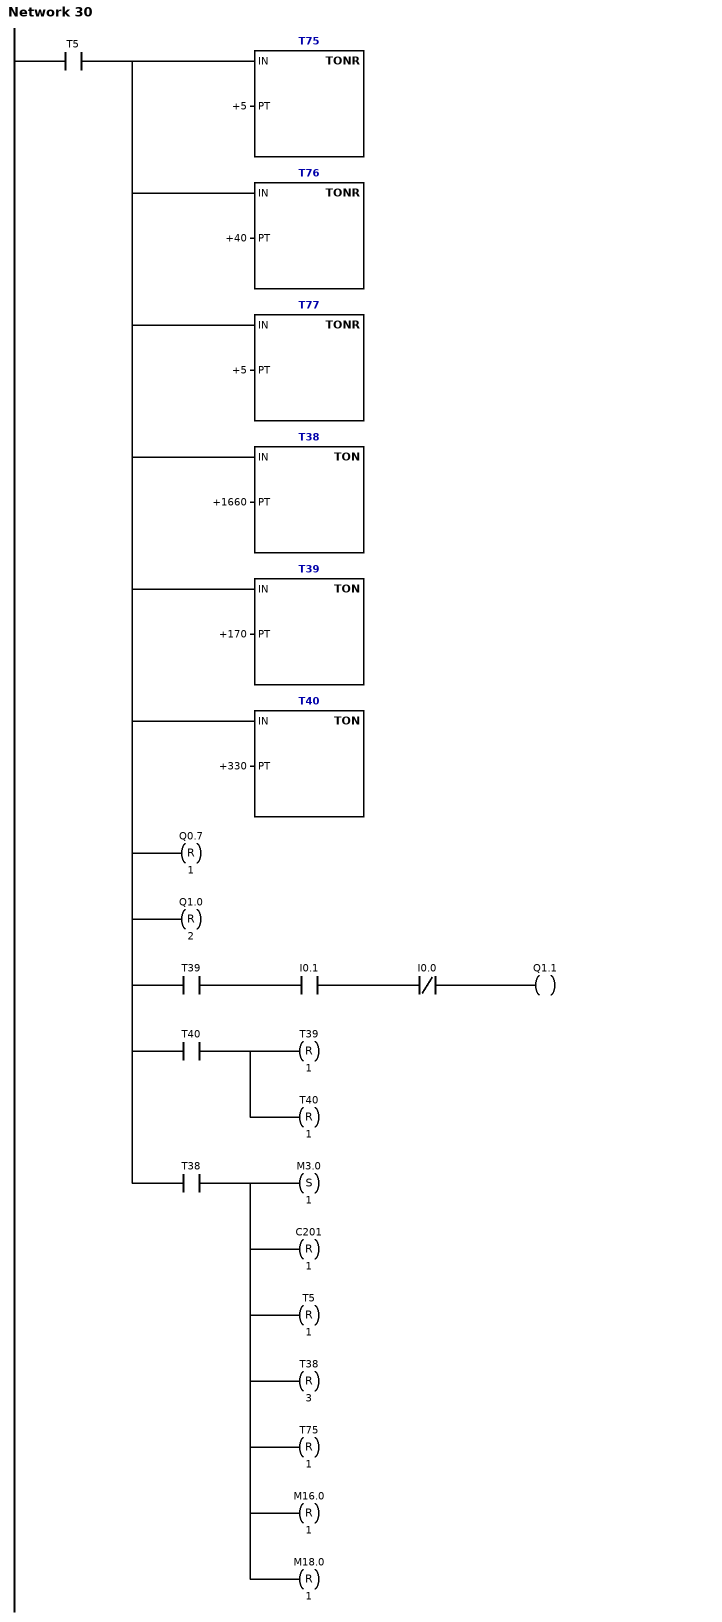
[picture p24: SBR4 networks 30-30]
Network 30
LD     T5
LPS
TONR   T75, +5
TONR   T76, +40
TONR   T77, +5
TON    T38, +1660
TON    T39, +170
TON    T40, +330
R      Q0.7, 1
R      Q1.0, 2
A      T39
A      I0.1
AN     I0.0
=      Q1.1
LRD
A      T40
R      T39, 1
R      T40, 1
LPP
A      T38
S      M3.0, 1
R      C201, 1
R      T5, 1
R      T38, 3
R      T75, 1
R      M16.0, 1
R      M18.0, 1
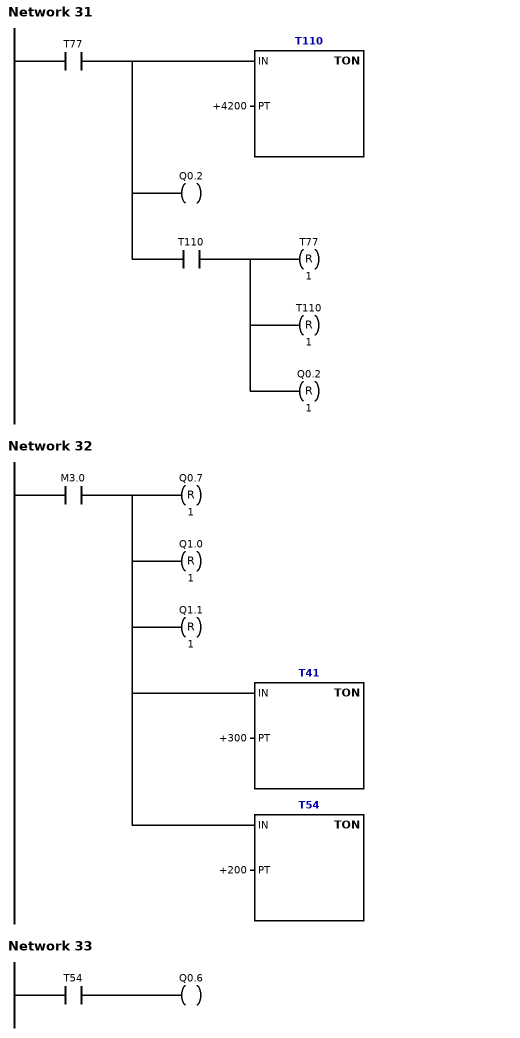
Network 31
LD     T77
TON    T110, +4200
=      Q0.2
A      T110
R      T77, 1
R      T110, 1
R      Q0.2, 1
Network 32
LD     M3.0
R      Q0.7, 1
R      Q1.0, 1
R      Q1.1, 1
TON    T41, +300
TON    T54, +200
Network 33
LD     T54
=      Q0.6
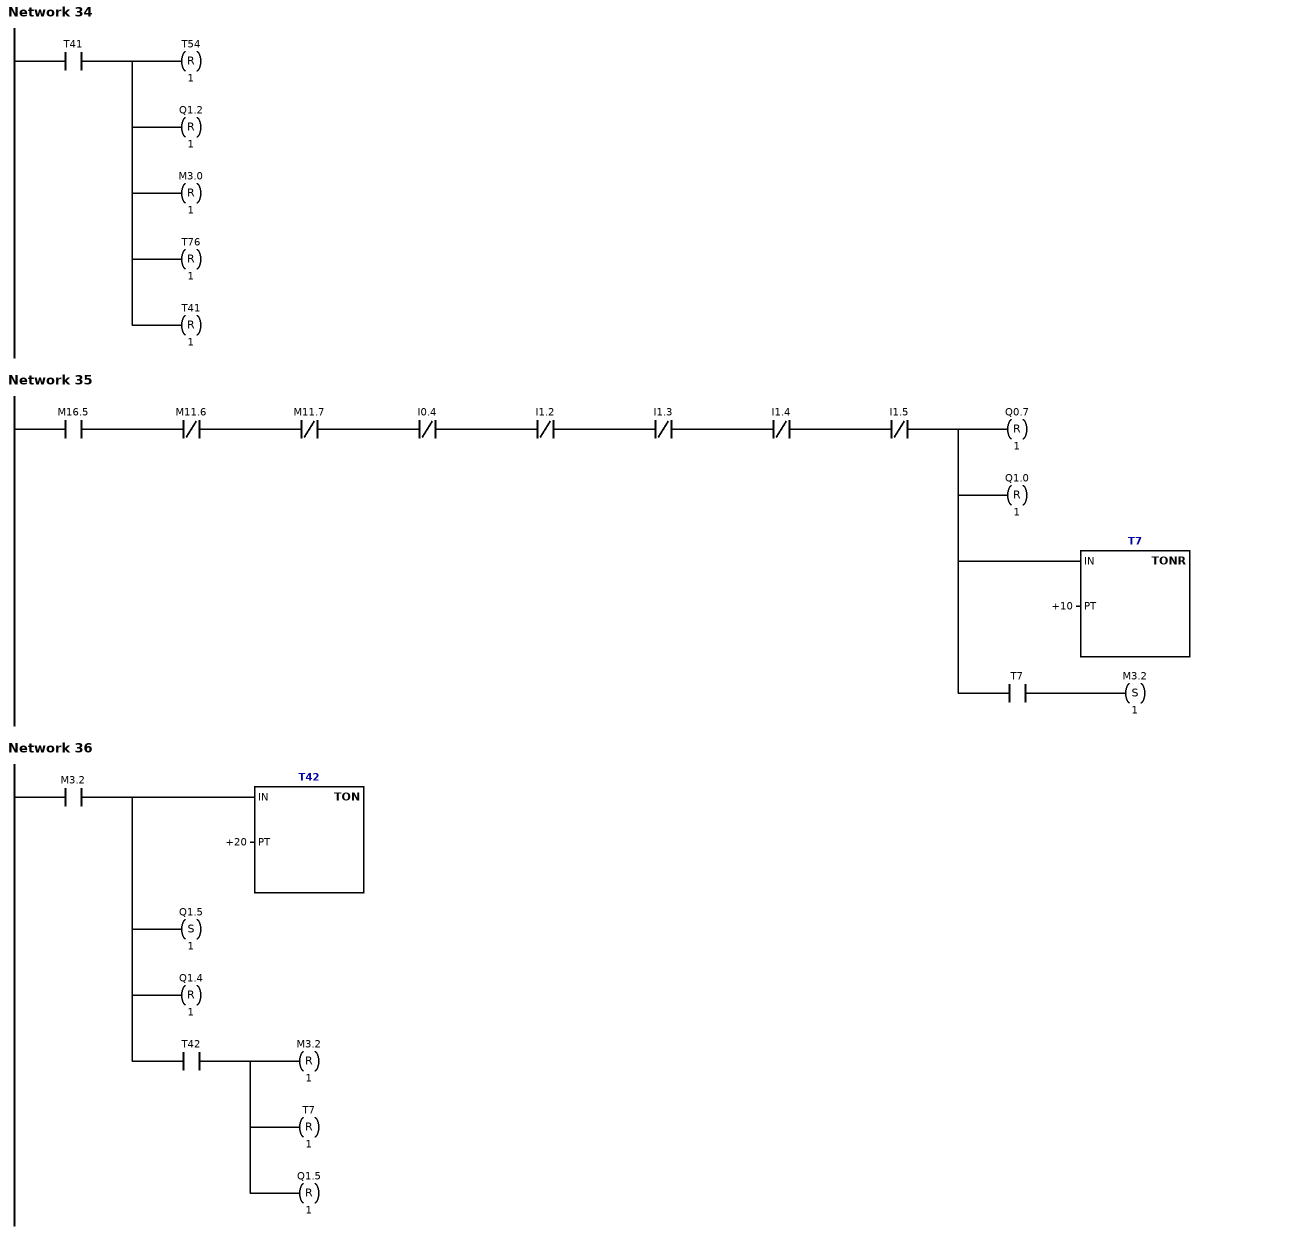
Network 34
LD     T41
R      T54, 1
R      Q1.2, 1
R      M3.0, 1
R      T76, 1
R      T41, 1
Network 35
LD     M16.5
AN     M11.6
AN     M11.7
AN     I0.4
AN     I1.2
AN     I1.3
AN     I1.4
AN     I1.5
R      Q0.7, 1
R      Q1.0, 1
TONR   T7, +10
A      T7
S      M3.2, 1
Network 36
LD     M3.2
TON    T42, +20
S      Q1.5, 1
R      Q1.4, 1
A      T42
R      M3.2, 1
R      T7, 1
R      Q1.5, 1
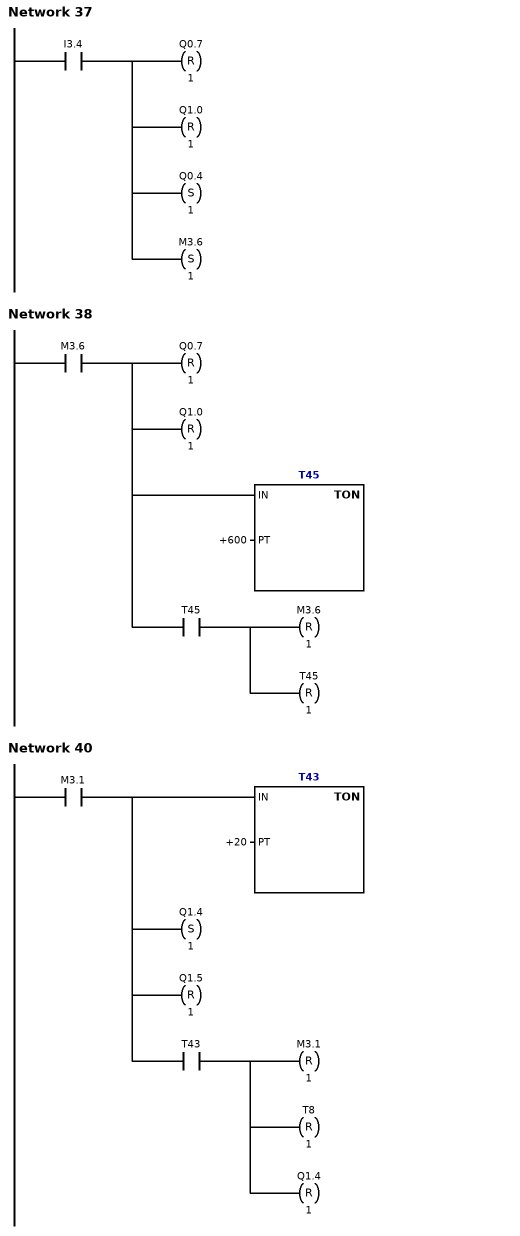
Network 37
LD     I3.4
R      Q0.7, 1
R      Q1.0, 1
S      Q0.4, 1
S      M3.6, 1
Network 38
LD     M3.6
R      Q0.7, 1
R      Q1.0, 1
TON    T45, +600
A      T45
R      M3.6, 1
R      T45, 1
Network 39
AN     M11.6
AN     M11.7
AN     I1.0
AN     I1.2
AN     I1.3
AN     I1.4
AN     I1.5
R      Q0.7, 1
R      Q1.0, 1
TONR   T8, +10
A      T8
S      M3.1, 1
Network 40
LD     M3.1
TON    T43, +20
S      Q1.4, 1
R      Q1.5, 1
A      T43
R      M3.1, 1
R      T8, 1
R      Q1.4, 1
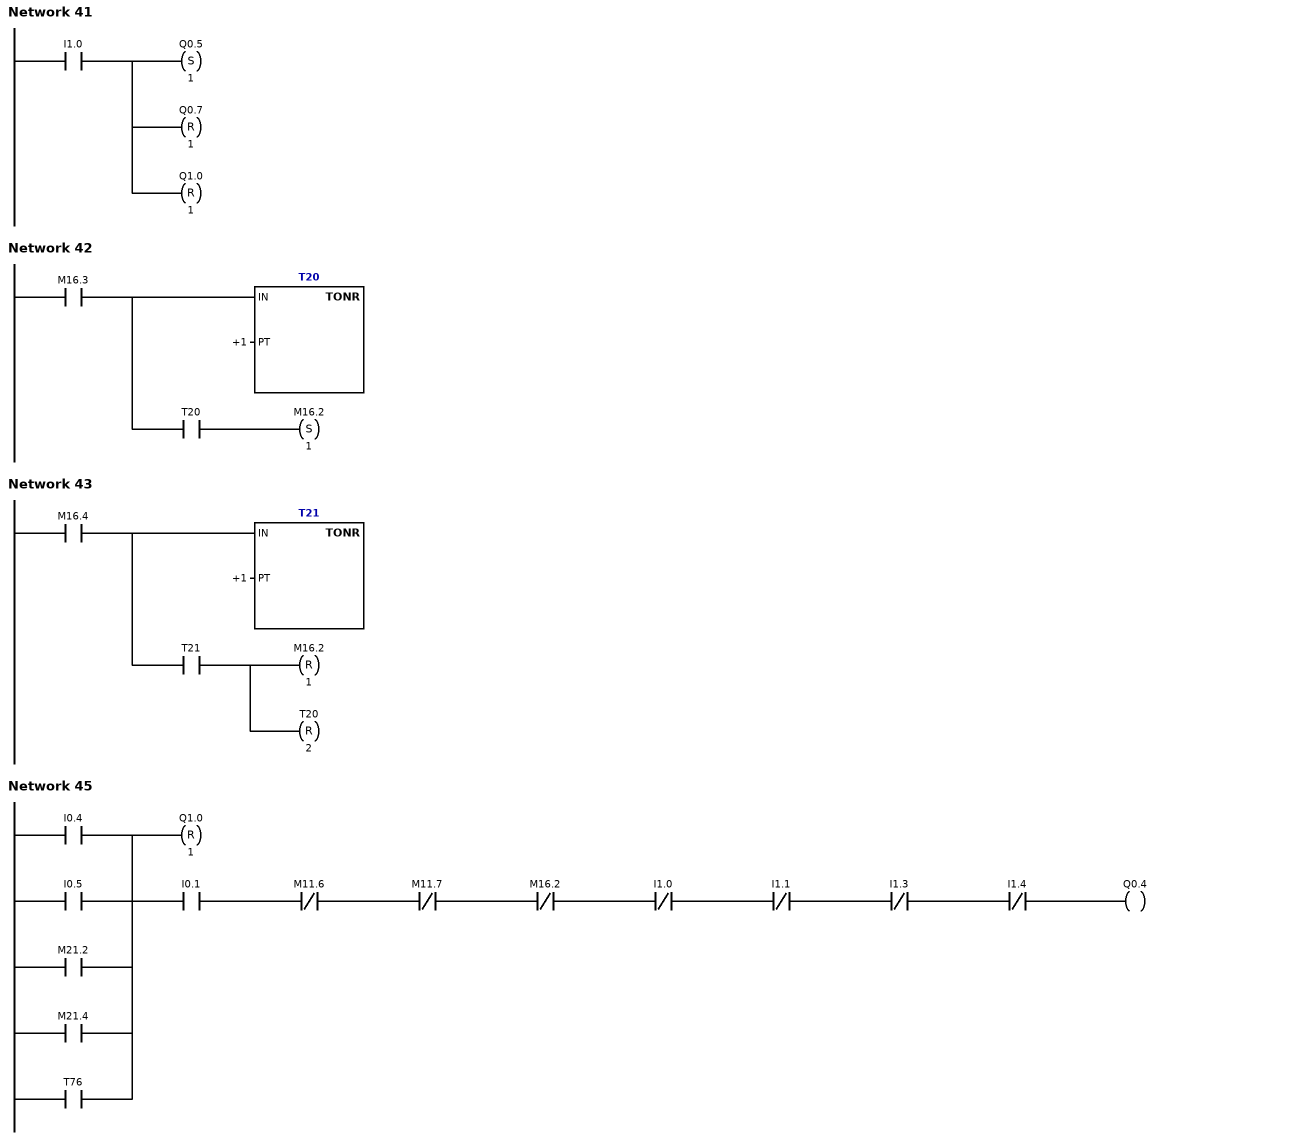
Network 41
LD     I1.0
S      Q0.5, 1
R      Q0.7, 1
R      Q1.0, 1
Network 42
LD     M16.3
TONR   T20, +1
A      T20
S      M16.2, 1
Network 43
LD     M16.4
TONR   T21, +1
A      T21
R      M16.2, 1
R      T20, 2
Network 45
LD     I0.4
O      I0.5
O      M21.2
O      M21.4
O      T76
R      Q1.0, 1
A      I0.1
AN     M11.6
AN     M11.7
AN     M16.2
AN     I1.0
AN     I1.1
AN     I1.3
AN     I1.4
=      Q0.4
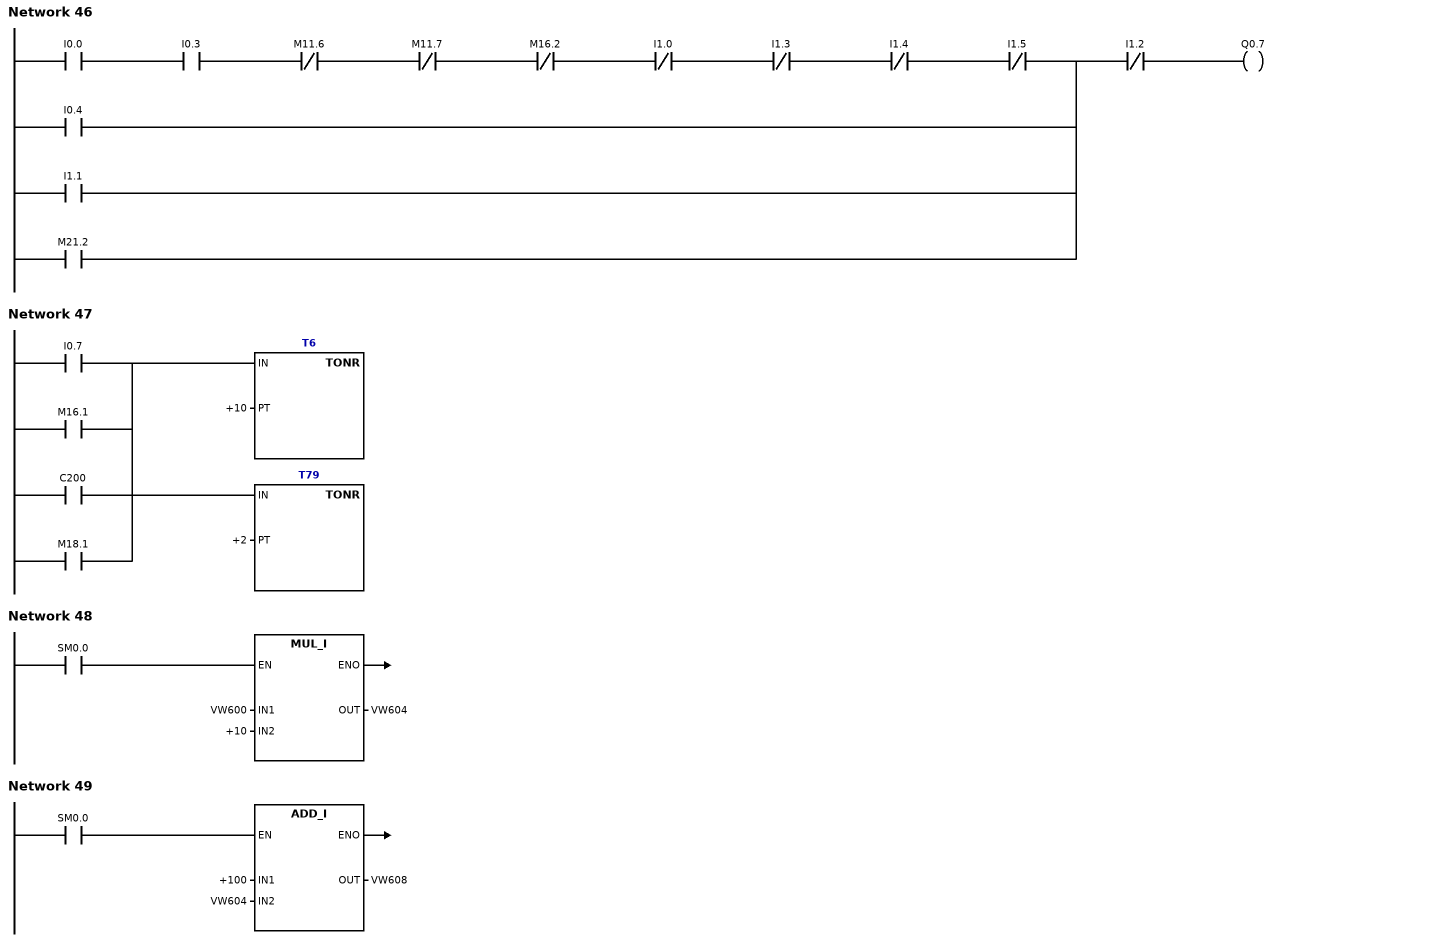
Network 46
LD     I0.0
A      I0.3
AN     M11.6
AN     M11.7
AN     M16.2
AN     I1.0
AN     I1.3
AN     I1.4
AN     I1.5
O      I0.4
O      I1.1
O      M21.2
AN     I1.2
=      Q0.7
Network 47
LD     I0.7
O      M16.1
O      C200
O      M18.1
TONR   T6, +10
TONR   T79, +2
Network 48
LD     SM0.0
MOVW   VW600, VW604
*I     +10, VW604
Network 49
LD     SM0.0
MOVW   +100, VW608
+I     VW604, VW608
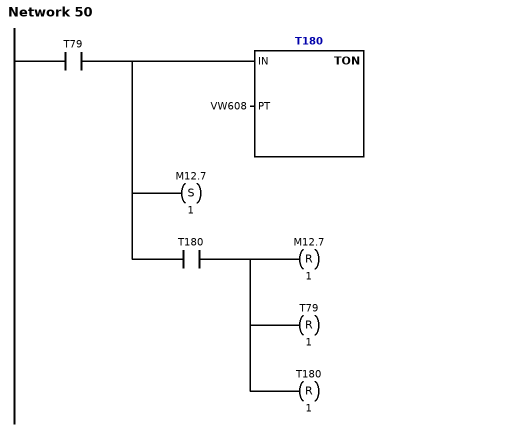
Network 50
LD     T79
TON    T180, VW608
S      M12.7, 1
A      T180
R      M12.7, 1
R      T79, 1
R      T180, 1
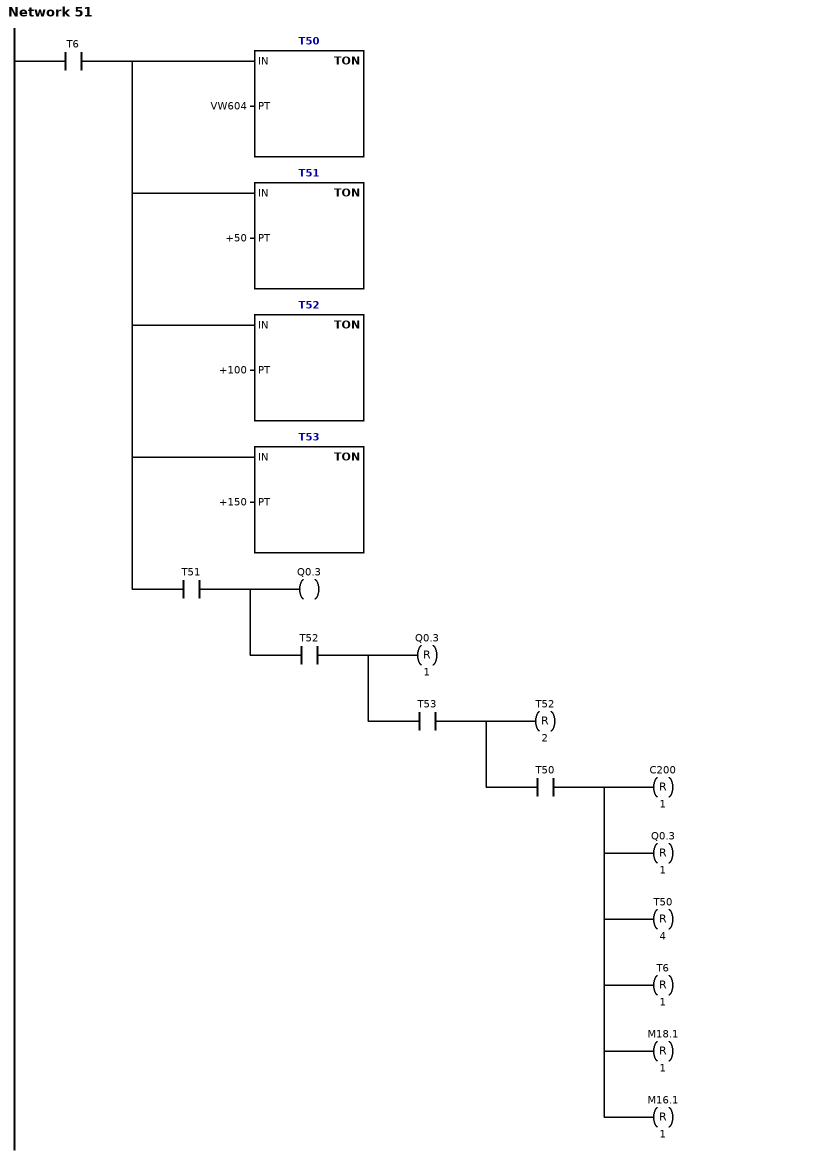
Network 51
LD     T6
TON    T50, VW604
TON    T51, +50
TON    T52, +100
TON    T53, +150
A      T51
=      Q0.3
A      T52
R      Q0.3, 1
A      T53
R      T52, 2
A      T50
R      C200, 1
R      Q0.3, 1
R      T50, 4
R      T6, 1
R      M18.1, 1
R      M16.1, 1
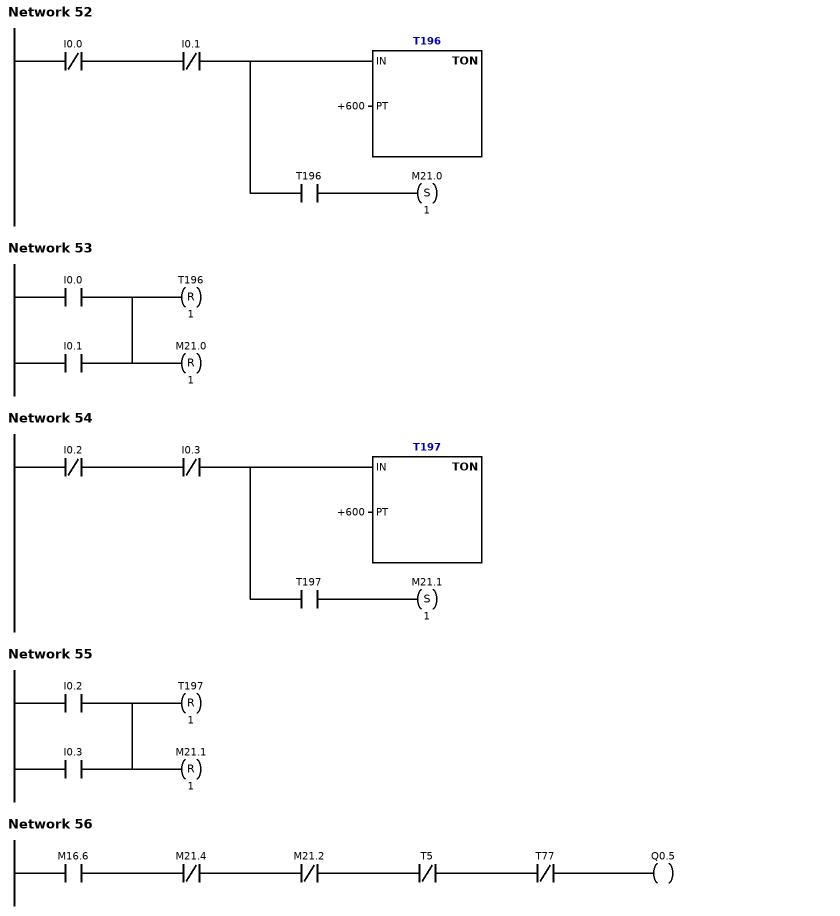
Network 52
LDN    I0.0
AN     I0.1
TON    T196, +600
A      T196
S      M21.0, 1
Network 53
LD     I0.0
O      I0.1
R      T196, 1
R      M21.0, 1
Network 54
LDN    I0.2
AN     I0.3
TON    T197, +600
A      T197
S      M21.1, 1
Network 55
LD     I0.2
O      I0.3
R      T197, 1
R      M21.1, 1
Network 56
LD     M16.6
AN     M21.4
AN     M21.2
AN     T5
AN     T77
=      Q0.5
END_SUBROUTINE_BLOCK

SUBROUTINE_BLOCK AutoRead:SBR5
TITLE=
BEGIN
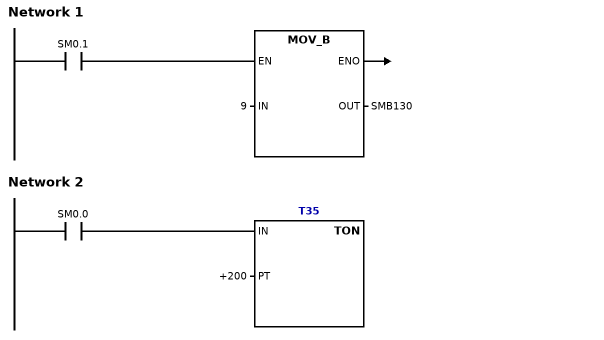
Network 1
LD     SM0.1
MOVB   9, SMB130
Network 2
LD     SM0.0
TON    T35, +200
Network 3
LD     T35
MOVB   58, VB300
MOVB   56, VB301
MOVB   56, VB302
MOVB   56, VB303
MOVB   56, VB304
MOVB   56, VB305
MOVB   56, VB306
MOVB   56, VB307
MOVB   48, VB308
MOVB   48, VB309
MOVB   48, VB310
MOVB   48, VB311
MOVB   51, VB312
MOVB   57, VB313
MOVB   52, VB314
MOVB   52, VB315
MOVB   50, VB316
MOVW   AIW4, VW317
MOVW   AIW6, VW319
MOVW   AIW16, VW321
MOVW   AIW18, VW323
MOVW   AIW8, VW325
MOVW   AIW10, VW327
MOVW   AIW12, VW329
MOVW   AIW14, VW331
MOVW   VW32, VW333
MOVW   VW30, VW335
MOVW   VW20, VW337
MOVW   VW80, VW339
MOVW   VW24, VW341
MOVW   VW82, VW343
MOVW   VW50, VW345
MOVW   VW22, VW347
MOVW   VW52, VW349
MOVW   VW26, VW351
MOVB   IB0, VB353
MOVB   IB1, VB354
MOVB   IB2, VB355
MOVB   QB0, VB356
MOVB   QB1, VB357
MOVB   QB2, VB358
MOVW   +0, T35
END_SUBROUTINE_BLOCK

SUBROUTINE_BLOCK Write2:SBR6
TITLE=
BEGIN
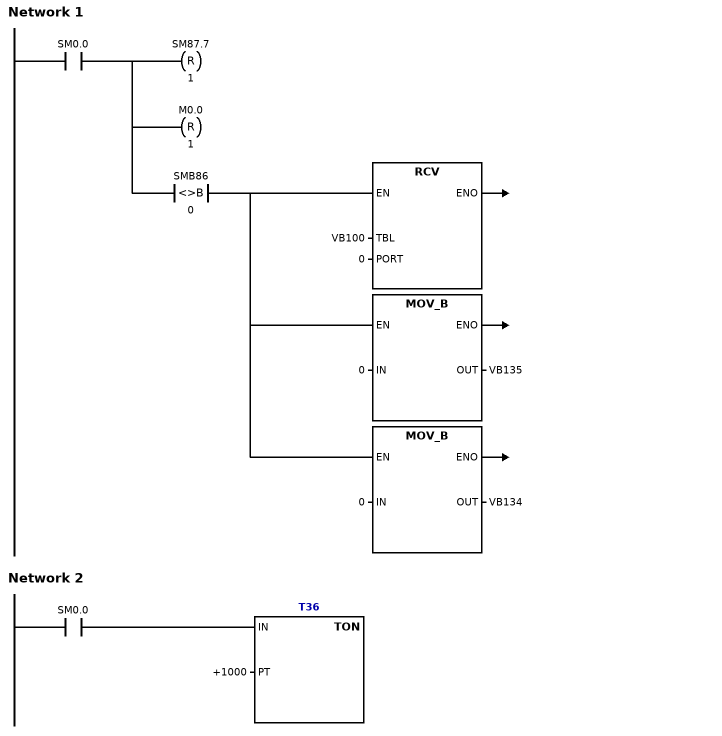
Network 1
LD     SM0.0
R      SM87.7, 1
R      M0.0, 1
AB<>   SMB86, 0
RCV    VB100, 0
MOVB   0, VB135
MOVB   0, VB134
Network 2
LD     SM0.0
TON    T36, +1000
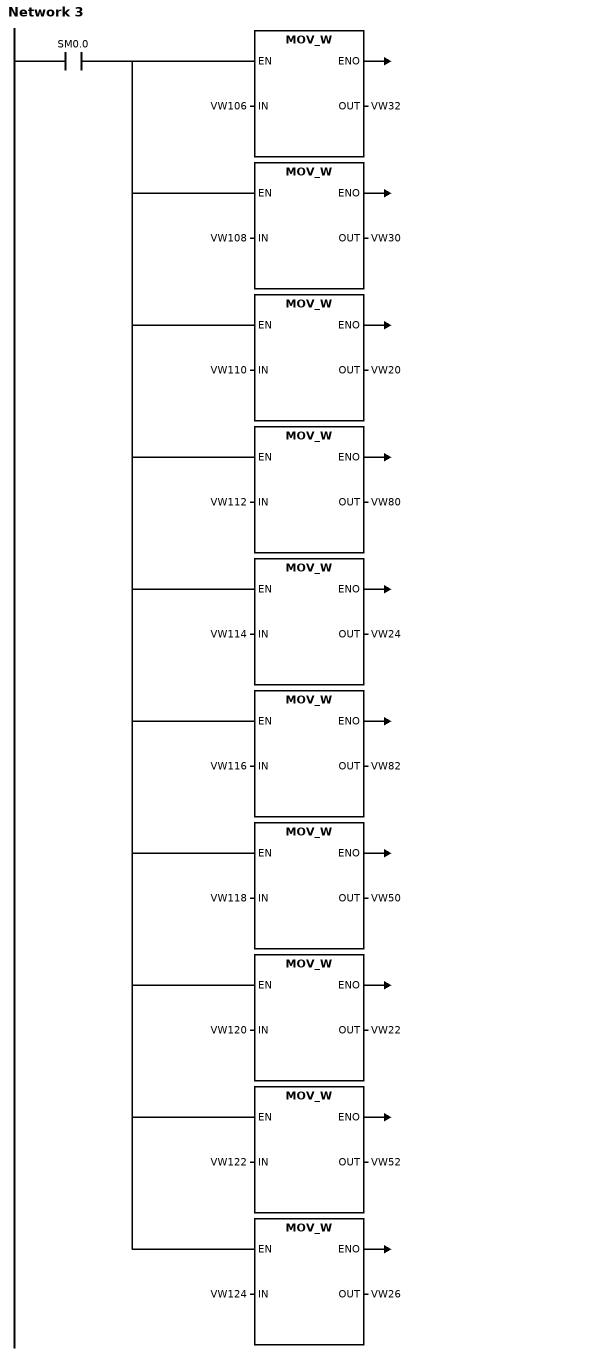
Network 3
LD     SM0.0
MOVW   VW106, VW32
MOVW   VW108, VW30
MOVW   VW110, VW20
MOVW   VW112, VW80
MOVW   VW114, VW24
MOVW   VW116, VW82
MOVW   VW118, VW50
MOVW   VW120, VW22
MOVW   VW122, VW52
MOVW   VW124, VW26
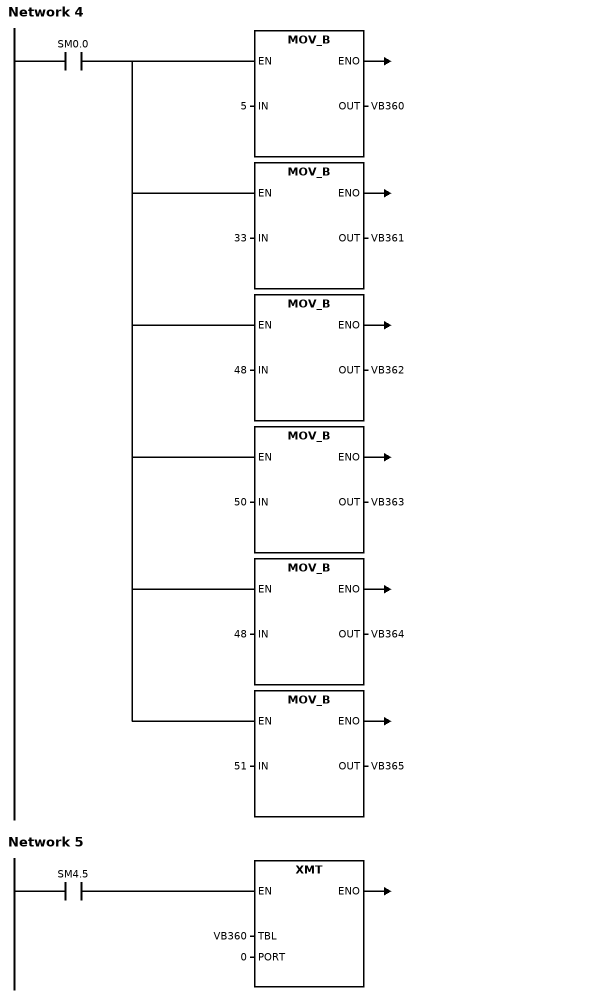
Network 4
LD     SM0.0
MOVB   5, VB360
MOVB   33, VB361
MOVB   48, VB362
MOVB   50, VB363
MOVB   48, VB364
MOVB   51, VB365
Network 5
LD     SM4.5
XMT    VB360, 0
END_SUBROUTINE_BLOCK

INTERRUPT_BLOCK RCVcomplete:INT0
TITLE=中断程序注释
BEGIN
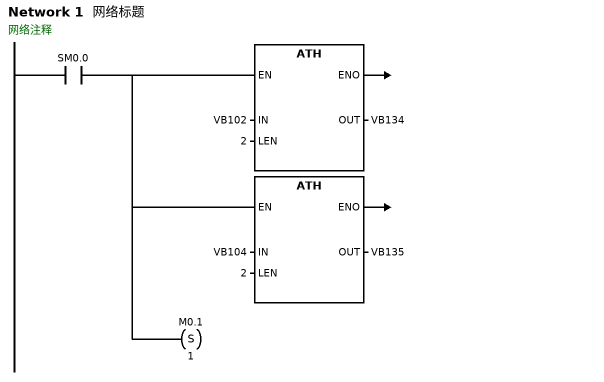
Network 1 // 网络标题
// 网络注释
LD     SM0.0
ATH    VB102, VB134, 2
ATH    VB104, VB135, 2
S      M0.1, 1
END_INTERRUPT_BLOCK

INTERRUPT_BLOCK XMTcomplete:INT1
TITLE=
BEGIN
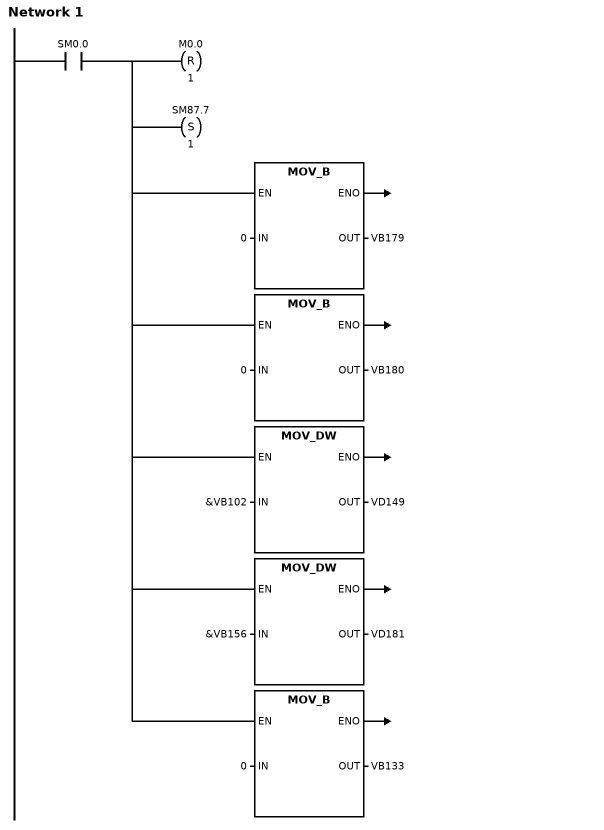
Network 1
LD     SM0.0
R      M0.0, 1
S      SM87.7, 1
MOVB   0, VB179
MOVB   0, VB180
MOVD   &VB102, VD149
MOVD   &VB156, VD181
MOVB   0, VB133
END_INTERRUPT_BLOCK

// (further data pages could not be read)
